// TIA Portal V19 export
DATA_BLOCK "DATE& TIME_DB"   // DB10
{ S7_Optimized_Access := 'TRUE' }
// stored: MemoryReserve 100
   VAR RETAIN
      READ : DTL;
      WRITE : DTL;
   END_VAR
   VAR
      SET : Bool;
      READ_DATE : Int;
      WRITE__DATE : Int;
   END_VAR
BEGIN
END_DATA_BLOCK
